{attribute 'GeneratedUsingTerminal: EP3632-0001-0016'}
{attribute addProperty BoxType "EP3632-0001-0016"}
{attribute addProperty Id "STATUSAT %I*STATUS_B07533568"}
{attribute addProperty CRC "1971471493"}
{attribute addProperty Size "8"}
TYPE Ch1_Status_75824485 EXTENDS InputBase_8311D824 :
STRUCT
	{attribute addProperty Name "STATUS"}
	STATUS AT %I* : STATUS_B0753356;
END_STRUCT
END_TYPE

(* stored: Version 1.2.0.0, ProductVersion 3.1.4024.11
   DUT Ch1_Status_75824485: Id {86ab84d3-fd60-4f6a-bdf0-5fe7586ae1de} *)
